// TIA Portal V20 export
DATA_BLOCK "CallEquipment_DB"   // DB59
{ DB_Accessible_From_OPC_UA := 'FALSE' }
// stored: AssignedProDiagFB Unit1.Em7.ProDiag, DBAccessibleFromOPCUA false, DBAccessibleFromWebserver false, InstanceOfName Unit1.Em7.CallEquipment, InstanceOfType FB, Namespace Unit1.Em7
"Unit1.Em7.CallEquipment"
   // VAR_INPUT
   //    ZoneOperationEnable { ExternalWritable := 'False'} : "LWONIK_typeSafetyZoneManualOperation";
   // END_VAR
   // VAR_IN_OUT
   //    unitStatus : "LAF_typeUnitStatus";
   //    emFeedback : "LUC_typeEmFeedback";
   //    unitAlarmDB : "LAF_typeAlarms";
   // END_VAR
   // VAR
   //    InstHotPressRightSequence { ExternalWritable := 'False'} : "Unit1.Em7.Sequence_1_HotPressRight";
   //    instHotPressRightHomeJob1 { ExternalWritable := 'False'} : "LAF_SelectJob";
   //    instHotPressRightLoadJob2 { ExternalWritable := 'False'} : "LAF_SelectJob";
   //    instHotPressRightInspectionJob3 { ExternalWritable := 'False'} : "LAF_SelectJob";
   //    instHotPressRightUnloadJob4 { ExternalWritable := 'False'} : "LAF_SelectJob";
   //    instCmHotPressRightSafetyPin { ExternalWritable := 'False'} : "LBC_DigitalSignalCn";
   //    instCmHotPressRightJRDetect { ExternalWritable := 'False'} : "LBC_DigitalSignalCn";
   //    instCmHotPressRightStageLiftFrontUpDown { ExternalWritable := 'False'} : "LBC_TwoWayActuatorCn";
   //    instCmHotPressRightStageLiftRearUpDown { ExternalWritable := 'False'} : "LBC_TwoWayActuatorCn";
   //    instCmHotPressRightStageLiftAllUpDown { ExternalWritable := 'False'} : "LBC_TwoWayActuatorCn";
   //    instCmHotPressRightTemperature { ExternalWritable := 'False'} : "LER_Heater";
   //    instCmHotPressRightServoPress { ExternalWritable := 'False'} : "LER_ServoPress";
   //    instCmHotPressRightHistroy { ExternalWritable := 'False'} : "LER_ServoPressHistory";
   //    instManageAlarms { ExternalWritable := 'False'} : "LAF_ManageAlarms";
   //    instEventsPFE { ExternalWritable := 'False'} : "Unit1.Em7.EventsPFE";
   //    statUnitStatus { ExternalWritable := 'False'} : "LAF_typeUnitStatus";
   //    statPartData { ExternalWritable := 'False'} : "LER_typePartData";
   //    statDataDelete { ExternalWritable := 'False'} : "LER_typePartData";
   //    statHistoryDeleteData { ExternalWritable := 'False'} : "LER_typeServoPressHistory";
   //    statClock { ExternalWritable := 'False'} : "LAF_typeGlobalClockMem";
   //    statTonTime { ExternalWritable := 'False'} : Array[0..999] of TON_TIME;
   //    statTofTime { ExternalWritable := 'False'} : Array[0..9] of TOF_TIME;
   //    statPulse { ExternalWritable := 'False'} : Array[0..999] of Bool;
   //    statNomalMode { ExternalWritable := 'False'} : Bool;
   //    statEnableManualCmds { ExternalWritable := 'False'} : Bool;
   //    statDoorOpenTemperature { ExternalWritable := 'False'} : "Safety.typeHotPressTempOk";
   //    statRunTemperature { ExternalWritable := 'False'} : Bool;
   //    "*** Interlock TwoWay ***" { S7_SetPoint := 'True'} : "LER_Axis_Homing";
   //    instCmHotPressRightStageLiftFrontUpDownInterlock { S7_SetPoint := 'True'} : Array[0..2] of "LER_Actuator";
   //    instCmHotPressRightStageLiftRearUpDownInterlock { S7_SetPoint := 'True'} : Array[0..2] of "LER_Actuator";
   //    instCmHotPressRightStageLiftAllUpDownInterlock { S7_SetPoint := 'True'} : Array[0..2] of "LER_Actuator";
   //    HotPressRightStageLiftFrontUpDown_Inpos : Array[0..2] of Struct
   //       "Int" : Array[1..10] of Bool;
   //    END_STRUCT;
   //    HotPressRightStageLiftRearUpDown_Inpos : Array[0..2] of Struct
   //       "Int" : Array[1..10] of Bool;
   //    END_STRUCT;
   //    HotPressRightStageLiftAllUpDown_Inpos : Array[0..2] of Struct
   //       "Int" : Array[1..10] of Bool;
   //    END_STRUCT;
   //    citi_Ptrig : Array[0..20] of Bool;
   //    citiTon : Array[0..20] of TON_TIME;
   //    citi : Time;
   //    citiTest : Array[0..20] of Bool;
   //    statReal : Array[0..9] of Real;
   //    instPFERecipe { S7_SetPoint := 'True'} : "Unit1.Em7.EventsPFE_Recipe";
   // END_VAR
BEGIN
END_DATA_BLOCK
